# B&R Automation Studio project Config_Logical
Automation Studio 4.9

## Logical view

Binary libraries used (declarations not repeated): operator, runtime, astime, AsIecCon, MpBase, CoTrace, AsZip, FileIO, McBase, McPathGen, MpAxis, MpPick, McAcpAx, McAxis, McProgInt, McAxGroup, MpRobotics, McAcpTrak 5.26.1, MpTool 5.26.1

### Global.var - Global variables
```iecst
VAR
	DeltaParameters : MpDelta4AxisParType;
	MpDelta4Axis_0 : MpDelta4Axis;
END_VAR

VAR CONSTANT
	P1 : McPointType := (Pos:=(X:=0, Y:=0, Z:=-650));
	P2 : McPointType := (Pos:=(X:=-50, Y:=-20, Z:=-600));
	P0 : McPointType := (Pos:=(X:=0, Y:=0, Z:=-560));
	P3 : McPointType := (Pos:=(X:=50, Y:=20, Z:=-540));
END_VAR
```


### Program Logical/Program (IEC)

#### Main.st
```iecst
PROGRAM _INIT

MpDelta4Axis_0.Enable := TRUE;

MpDelta4Axis_0.Override := 100.0;
DeltaParameters.ProgramName := 'Robotic.st';    //File stored on FileDevice

END_PROGRAM

PROGRAM _CYCLIC
gAxisQ4;
MpDelta4Axis_0.MpLink := ADR(g4AxDeltaA);
MpDelta4Axis_0.Parameters := ADR(DeltaParameters);
MpDelta4Axis_0();

END_PROGRAM
```

### Program Logical/PickAndPlace/PrgMechs

#### Types.typ
```iecst
TYPE
	RCStepEnum :
		(
		RC_WAIT_ENABLE,
		RC_POWER_ROBOT,
		RC_HOME_ROBOT,
		RC_ROBOT_READY,
		RC_WAIT_ENABLE_AXIS_FB,
		RC_POWER_AXIS,
		RC_WAIT_POWER_AXIS,
		RC_HOME_AXIS,
		RC_WAIT_HOME_AXIS,
		RC_READY,
		RC_START_PROCESS,
		RC_WAIT_PROCESS_STARTED,
		RC_PROCESSING,
		RC_ERROR,
		RC_ERROR_STOP
		);
END_TYPE
```

#### Main.st
```iecst
PROGRAM _INIT

    MpDelta4Axis_0.Override := 100.0;
    MpDelta4Axis_0.Enable   := TRUE;

    AxisParameters_0.Velocity     := 130.0;
    AxisParameters_0.Acceleration := 50.0;
    AxisParameters_0.Deceleration := 50.0;

    AxisParameters_1.Velocity     := 130.0;
    AxisParameters_1.Acceleration := 50.0;
    AxisParameters_1.Deceleration := 50.0;

    MpAxisBasic_0.Enable := TRUE;
    MpAxisBasic_1.Enable := TRUE;

    // dummy call of axis PVs just to avoid warning -2141192189 "The PV 'gAxisQx' does not exists" in logger
    gAxisQ1;
    gAxisQ2;
    gAxisQ3;
    gAxisQ4;

END_PROGRAM

PROGRAM _CYCLIC

    (* Prepare mechanics: Robot & conveyors *)
    CASE RC_Step OF

        (* first preparing robot *)
        RC_WAIT_ENABLE:
            IF MpDelta4Axis_0.Active THEN
                RC_Step := RC_POWER_ROBOT;
            END_IF

        RC_POWER_ROBOT:
            MpDelta4Axis_0.Power := TRUE;
            IF MpDelta4Axis_0.PowerOn THEN
                RC_Step := RC_HOME_ROBOT;
            END_IF

        RC_HOME_ROBOT:
           MpDelta4Axis_0.Home := TRUE;
           IF MpDelta4Axis_0.IsHomed THEN
                MpDelta4Axis_0.Home := FALSE;
                RC_Step := RC_ROBOT_READY;
           END_IF

        RC_ROBOT_READY:
            RC_Step := RC_WAIT_ENABLE_AXIS_FB;

        (* preparing conveyors *)
        RC_WAIT_ENABLE_AXIS_FB:
            IF MpAxisBasic_0.Active THEN
                IF MpAxisBasic_1.Active THEN
                    RC_Step := RC_POWER_AXIS;
                END_IF
            ELSIF MpAxisBasic_0.Error OR MpAxisBasic_1.Error THEN
                LastStep := RC_Step;
                RC_Step  := RC_ERROR;
            END_IF;

        RC_POWER_AXIS:
            MpAxisBasic_0.Power := TRUE;
            MpAxisBasic_1.Power := TRUE;
            RC_Step := RC_WAIT_POWER_AXIS;

        RC_WAIT_POWER_AXIS:
            IF MpAxisBasic_0.PowerOn THEN
                IF MpAxisBasic_1.PowerOn THEN
                    RC_Step := RC_HOME_AXIS;
                END_IF
            ELSIF MpAxisBasic_0.Error OR MpAxisBasic_1.Error THEN
                LastStep := RC_Step;
                RC_Step  := RC_ERROR;
            END_IF;

        RC_HOME_AXIS:
            MpAxisBasic_0.Home := TRUE;
            MpAxisBasic_1.Home := TRUE;
            RC_Step := RC_WAIT_HOME_AXIS;

        RC_WAIT_HOME_AXIS:
            IF MpAxisBasic_0.IsHomed THEN
                IF MpAxisBasic_0.IsHomed THEN
                    MpAxisBasic_0.Home := FALSE;
                    MpAxisBasic_1.Home := FALSE;
                    RC_Step := RC_READY;
                END_IF
            ELSIF MpAxisBasic_0.Error OR MpAxisBasic_1.Error THEN
                LastStep := RC_Step;
                RC_Step  := RC_ERROR;
            END_IF;

        RC_READY:
            ReadyMechanics := TRUE;
            IF CmdStart AND ReadyToStart THEN
                RC_Step := RC_START_PROCESS;
            END_IF;

        (* start conveyors to move *)
        RC_START_PROCESS:
            MpAxisBasic_0.MoveVelocity := TRUE;
            MpAxisBasic_1.MoveVelocity := TRUE;
            RC_Step := RC_WAIT_PROCESS_STARTED;

        RC_WAIT_PROCESS_STARTED:
            IF MpAxisBasic_0.Info.PLCopenState = mcAXIS_CONTINUOUS_MOTION THEN
                IF MpAxisBasic_1.Info.PLCopenState = mcAXIS_CONTINUOUS_MOTION THEN
                    RC_Step := RC_PROCESSING;
                END_IF
            ELSIF MpAxisBasic_0.Error OR MpAxisBasic_1.Error THEN
                LastStep := RC_Step;
                RC_Step  := RC_ERROR;
            END_IF;

        RC_PROCESSING:
            IF MpAxisBasic_0.Error OR MpAxisBasic_1.Error THEN
                LastStep := RC_Step;
                RC_Step  := RC_ERROR;
            END_IF;

        RC_ERROR:
            ReadyMechanics := FALSE;

    END_CASE

    ReadyToStart := ReadyMechanics AND ReadyPickReg AND ReadyPlaceReg AND ReadyPickCore;

    (* Call FBs *)
    MpDelta4Axis_0.MpLink     := ADR(g4AxDeltaA);
    MpDelta4Axis_0.Parameters := ADR(DeltaParameters);
    MpDelta4Axis_0();

    MpAxisBasic_0.MpLink     := ADR(gAxis_1);
    MpAxisBasic_0.Parameters := ADR(AxisParameters_0);
    MpAxisBasic_0();

    MpAxisBasic_1.MpLink     := ADR(gAxis_2);
    MpAxisBasic_1.Parameters := ADR(AxisParameters_1);
    MpAxisBasic_1();

    PickConveyorPosition  := MpAxisBasic_0.Position;
    PlaceConveyorPosition := MpAxisBasic_1.Position;

END_PROGRAM
```

### Program Logical/PickAndPlace/PrgPick

#### Variables.var
```iecst
VAR
	C_Step : ConvStepEnum;
	LastStep : ConvStepEnum;
	Error : BOOL;
	ProductSpacing : LREAL;
	LastProductConveyorPosition : LREAL;
	ElapsedDistance : LREAL;
END_VAR
(*  *)
(*Functionblocks*)
VAR
	MpPickRegister_0 : MpPickRegister;
	MpPickRegCreateProduct : MpPickRegCreateObject;
END_VAR
```

#### Main.st
```iecst
PROGRAM _INIT

    C_Step := C_WAIT_ENABLE;
    Error := FALSE;

    ProductSpacing := 120; // distance between two consecutive products

END_PROGRAM

PROGRAM _CYCLIC

    CASE C_Step OF
        C_WAIT_ENABLE:
            LastStep := C_WAIT_ENABLE;
            C_Step   := C_ENABLE_REGISTER_FB;

        (* Pick-and-Place register handling for Picking conveyor *)
        C_ENABLE_REGISTER_FB:
            MpPickRegister_0.Enable := TRUE;
            C_Step := C_WAIT_ENABLE_REGISTER_FB;

        C_WAIT_ENABLE_REGISTER_FB:
            IF MpPickRegister_0.Active THEN
                C_Step := C_ENABLE_REGISTER;
            ELSIF MpPickRegister_0.Error THEN
                LastStep := C_Step;
                C_Step   := C_ERROR;
            END_IF;

        C_ENABLE_REGISTER:
            MpPickRegister_0.RegisterEnable := TRUE;
            C_Step := C_WAIT_ENABLE_REGISTER;

        C_WAIT_ENABLE_REGISTER:
            IF MpPickRegister_0.RegisterActive THEN
                C_Step := C_ENABLE_ADD_REGISTER_FBS;
            ELSIF MpPickRegister_0.Error THEN
                LastStep := C_Step;
                C_Step   := C_ERROR;
            END_IF;

        C_ENABLE_ADD_REGISTER_FBS:
            MpPickRegCreateProduct.Enable := TRUE;
            C_Step := C_WAIT_ENABLE_ADD_REGISTER_FBS;

        C_WAIT_ENABLE_ADD_REGISTER_FBS:
            IF MpPickRegCreateProduct.Active THEN
                C_Step := C_WAIT_START_PROCESS;
            ELSIF MpPickRegCreateProduct.Error THEN
                LastStep := C_Step;
                C_Step   := C_ERROR;
            END_IF;

        C_WAIT_START_PROCESS: // waits user start command and conveyor moving
            ReadyPickReg := TRUE;
            IF CmdStart AND ReadyToStart AND (PickConveyorPosition > 0) THEN
                C_Step := C_PROCESSING;
            END_IF;

        C_PROCESSING: (* now create products on moving conveyor for picking *)

            ElapsedDistance := DistanceOverPeriod(PickConveyorPosition, LastProductConveyorPosition, PickConveyorLength);

            IF (ElapsedDistance >= ProductSpacing) THEN

                MpPickRegCreateProduct.Parameters.LatchedConveyor.Position:= PickConveyorPosition;
                MpPickRegCreateProduct.Parameters.Mode := mpPICK_CREATE_SINGLEITEM;
                MpPickRegCreateProduct.Parameters.ObjectTypeName := 'MyProduct';
                MpPickRegCreateProduct.Parameters.Translation.X  := 0;
                MpPickRegCreateProduct.Parameters.Translation.Y  := 125; // in the middle of conveyor width
                MpPickRegCreateProduct.Create := TRUE;

                LastProductConveyorPosition := MpPickRegCreateProduct.Parameters.LatchedConveyor.Position;
            ELSE
                MpPickRegCreateProduct.Create := FALSE;
            END_IF

            IF MpPickRegCreateProduct.Error THEN
                LastStep := C_Step;
                C_Step   := C_ERROR;
            END_IF;

        C_ERROR:
            Error := TRUE;
            ReadyPickReg := FALSE;

    END_CASE

    (* FB calls *)
    MpPickRegister_0.MpLink := ADR(gPickRegister);
    MpPickRegister_0();

    MpPickRegCreateProduct.MpLink := ADR(gPickRegister);
    MpPickRegCreateProduct();

END_PROGRAM
```

### Types.typ
```iecst
TYPE
	PickCoreStepEnum :
		(
		PC_WAIT_ENABLE,
		PC_ENABLE_PICK_CORE,
		PC_WAIT_ENABLE_PICK_CORE,
		PC_ENABLE_CORE_PROCESS,
		PC_WAIT_ENABLE_CORE_PROCESS,
		PC_WAIT_START_CORE_PROCESS,
		PC_READY_TO_START,
		PC_STARTED,
		PC_ERROR
		);
END_TYPE
```

### Program Logical/PickAndPlace/PrgPlace

#### Variables.var
```iecst
VAR
	P_Step : PlaceStepEnum;
	LastStep : PlaceStepEnum;
	Error : BOOL;
	PlaceHoldersSpacing : LREAL;
	LastPlaceHolderConveyorPosition : LREAL;
	ElapsedDistance : LREAL;
END_VAR
(*   *)
(*Functionblocks*)
VAR
	MpPickRegister_0 : MpPickRegister;
	MpPickRegCreatePlaceholder : MpPickRegCreateObject;
END_VAR
```

#### Main.st
```iecst
PROGRAM _INIT

    P_Step := P_WAIT_ENABLE;
    Error := FALSE;

    PlaceHoldersSpacing := 120; // distance between two consecutive place holders

END_PROGRAM

PROGRAM _CYCLIC

    CASE P_Step OF
        P_WAIT_ENABLE:
            P_Step := P_ENABLE_REGISTER_FB;

        P_ENABLE_REGISTER_FB:
            MpPickRegister_0.Enable := TRUE;
            P_Step := P_WAIT_ENABLE_REGISTER_FB;

        P_WAIT_ENABLE_REGISTER_FB:
            IF MpPickRegister_0.Active THEN
                P_Step := P_ENABLE_REGISTER_COMP;

            ELSIF MpPickRegister_0.Error THEN
                LastStep := P_Step;
                P_Step := P_ERROR;
            END_IF;

        P_ENABLE_REGISTER_COMP:
            MpPickRegister_0.RegisterEnable := TRUE;
            P_Step := P_WAIT_ENABLE_REGISTER_COMP;

        P_WAIT_ENABLE_REGISTER_COMP:
            IF MpPickRegister_0.RegisterActive THEN
                P_Step := P_ENABLE_ADD_REGISTER_FBS;

            ELSIF MpPickRegister_0.Error THEN
                LastStep := P_Step;
                P_Step := P_ERROR;
            END_IF;

        P_ENABLE_ADD_REGISTER_FBS:
            MpPickRegCreatePlaceholder.Enable := TRUE;
            MpPickRegCreatePlaceholder.Create := FALSE;
            P_Step := P_WAIT_ENABLE_ADD_REGISTER_FBS;

        P_WAIT_ENABLE_ADD_REGISTER_FBS:
            IF 	MpPickRegCreatePlaceholder.Active THEN
                P_Step := P_WAIT_START_PROCESS;

            ELSIF MpPickRegCreatePlaceholder.Error THEN
                LastStep := P_Step;
                P_Step := P_ERROR;
            END_IF;

        P_WAIT_START_PROCESS: // waits user start command and conveyor moving
            ReadyPlaceReg := TRUE;
            IF CmdStart AND ReadyToStart AND (PlaceConveyorPosition > 0) THEN
                P_Step := P_CREATE_OBJECTS;
            END_IF;

        (* We need to create positions (place holders) on place conveyor where to place picked objects *)
        P_CREATE_OBJECTS:

            ElapsedDistance := DistanceOverPeriod(PlaceConveyorPosition, LastPlaceHolderConveyorPosition, PlaceConveyorLength);

            IF (ElapsedDistance >= PlaceHoldersSpacing) THEN

                MpPickRegCreatePlaceholder.Parameters.LatchedConveyor.Position := PlaceConveyorPosition;
                MpPickRegCreatePlaceholder.Parameters.Mode := mpPICK_CREATE_SINGLEITEM_PLACEH;
                MpPickRegCreatePlaceholder.Parameters.ObjectTypeName := 'MyProduct';
                MpPickRegCreatePlaceholder.Parameters.Translation.X := 0;
                MpPickRegCreatePlaceholder.Parameters.Translation.Y := 125; // in the middle of conveyor width
                MpPickRegCreatePlaceholder.Create := TRUE;

                LastPlaceHolderConveyorPosition := MpPickRegCreatePlaceholder.Parameters.LatchedConveyor.Position;
            ELSE
                MpPickRegCreatePlaceholder.Create := FALSE;
            END_IF

        P_ERROR:
            Error := TRUE;
            ReadyPlaceReg := FALSE;

    END_CASE;

    (* FB calls *)
    MpPickRegister_0.MpLink := ADR(gPlaceRegister);
    MpPickRegister_0();

    MpPickRegCreatePlaceholder.MpLink := ADR(gPlaceRegister);
	MpPickRegCreatePlaceholder();

END_PROGRAM
```

Listed in the project but not available here: Logical/Global.typ, Logical/Robotic.st
